// TIA Portal V17 export
// export: Created 2025-03-05T08:00:44.5361321Z, ExportSetting WithDefaults, DisplayName Totally Integrated Automation Portal, DisplayVersion V17 Update 8, DisplayName TIA Portal Openness, DisplayVersion V17 Update 8, DisplayName TIA Portal Version Control Interface, DisplayVersion V17, DisplayName SINAMICS Startdrive Advanced, DisplayVersion V17 SP2, DisplayName SINAMICS Startdrive G110M, G120, G120C, G120D, G120P, G115D, DisplayVersion V17 SP2, DisplayName SINAMICS Startdrive G130, G150, S120, S150, SINAMICS MV, S210, DisplayVersion V17 SP2, DisplayName STEP 7 Professional, DisplayVersion V17 Update 8, DisplayName SINUMERIK ONE STEP 7 Toolbox, DisplayVersion V17 Update 12, DisplayName SINUMERIK 840D sl STEP 7 Toolbox, DisplayVersion V17 Update 12, DisplayName STEP 7 Safety, DisplayVersion V17 Update 6, DisplayName WinCC Advanced, DisplayVersion V17 Update 8
FUNCTION "FC1314_UNIT_03_MASTER_MEASUREMENT" : Void   // FC1314, LAD
{ S7_Optimized_Access := 'FALSE' }
AUTHOR : ETXETAR
VERSION : 1.0
// stored: AutoNumber false, IsIECCheckEnabled false, SetENOAutomatically false, UDAEnableTagReadback false
   VAR_TEMP
      UNIT_01_STATION_0_LOCAL_E_RETURNS : Bool;   // UNIT 01 STATION 0 LOCAL E RETURNS
      UNIT_01_STATION_0_MACHINE_E_RETURNS : Bool;   // UNIT 01 STATION 0 MACHINE E RETURNS
   END_VAR
   VAR CONSTANT
      FC_NUMBER : DInt := 1314;
   END_VAR
   VAR_TEMP   // added for the SCL form of the ladder/FBD networks
      _w1 : Bool;
   END_VAR
BEGIN

REGION Network 1: GENERAL CONDITIONS
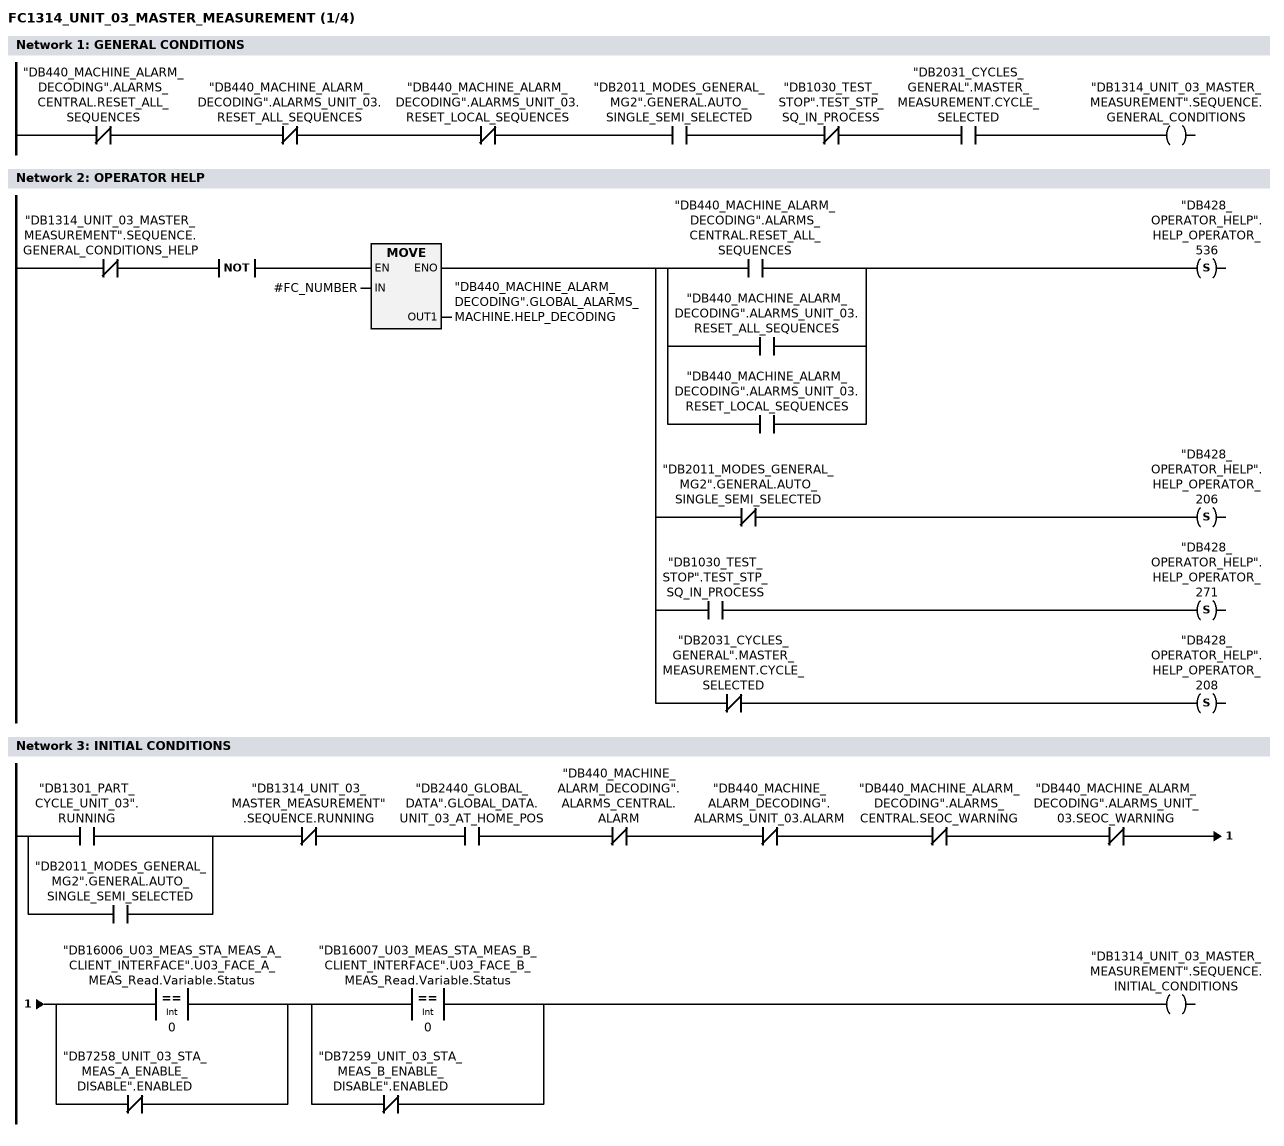
   RUNG wire#powerrail
      I_Contact( "DB440_MACHINE_ALARM_DECODING".ALARMS_CENTRAL.RESET_ALL_SEQUENCES )
      I_Contact( "DB440_MACHINE_ALARM_DECODING".ALARMS_UNIT_03.RESET_ALL_SEQUENCES )
      I_Contact( "DB440_MACHINE_ALARM_DECODING".ALARMS_UNIT_03.RESET_LOCAL_SEQUENCES )
      Contact( "DB2011_MODES_GENERAL_MG2".GENERAL.AUTO_SINGLE_SEMI_SELECTED )
      I_Contact( "DB1030_TEST_STOP".TEST_STP_SQ_IN_PROCESS )
      Contact( "DB2031_CYCLES_GENERAL".MASTER_MEASUREMENT.CYCLE_SELECTED )
      Coil( "DB1314_UNIT_03_MASTER_MEASUREMENT".SEQUENCE.GENERAL_CONDITIONS )
   END_RUNG
   // the same network as SCL:
   "DB1314_UNIT_03_MASTER_MEASUREMENT".SEQUENCE.GENERAL_CONDITIONS := NOT "DB440_MACHINE_ALARM_DECODING".ALARMS_CENTRAL.RESET_ALL_SEQUENCES AND NOT "DB440_MACHINE_ALARM_DECODING".ALARMS_UNIT_03.RESET_ALL_SEQUENCES AND NOT "DB440_MACHINE_ALARM_DECODING".ALARMS_UNIT_03.RESET_LOCAL_SEQUENCES AND "DB2011_MODES_GENERAL_MG2".GENERAL.AUTO_SINGLE_SEMI_SELECTED AND NOT "DB1030_TEST_STOP".TEST_STP_SQ_IN_PROCESS AND "DB2031_CYCLES_GENERAL".MASTER_MEASUREMENT.CYCLE_SELECTED;
END_REGION

REGION Network 2: OPERATOR HELP
   RUNG wire#powerrail
      I_Contact( "DB1314_UNIT_03_MASTER_MEASUREMENT".SEQUENCE.GENERAL_CONDITIONS_HELP )
      Not()
      { S7_GenerateENO := "TRUE" } Move(in := #FC_NUMBER, out1 => "DB440_MACHINE_ALARM_DECODING".GLOBAL_ALARMS_MACHINE.HELP_DECODING)
      wire#w1
      Contact( "DB440_MACHINE_ALARM_DECODING".ALARMS_CENTRAL.RESET_ALL_SEQUENCES )
      wire#w2
      S_Coil( "DB428_OPERATOR_HELP".HELP_OPERATOR_536 )
   END_RUNG
   RUNG wire#w1
      Contact( "DB440_MACHINE_ALARM_DECODING".ALARMS_UNIT_03.RESET_ALL_SEQUENCES )
   END_RUNG wire#w2
   RUNG wire#w1
      Contact( "DB440_MACHINE_ALARM_DECODING".ALARMS_UNIT_03.RESET_LOCAL_SEQUENCES )
   END_RUNG wire#w2
   RUNG wire#w1
      I_Contact( "DB2011_MODES_GENERAL_MG2".GENERAL.AUTO_SINGLE_SEMI_SELECTED )
      S_Coil( "DB428_OPERATOR_HELP".HELP_OPERATOR_206 )
   END_RUNG
   RUNG wire#w1
      Contact( "DB1030_TEST_STOP".TEST_STP_SQ_IN_PROCESS )
      S_Coil( "DB428_OPERATOR_HELP".HELP_OPERATOR_271 )
   END_RUNG
   RUNG wire#w1
      I_Contact( "DB2031_CYCLES_GENERAL".MASTER_MEASUREMENT.CYCLE_SELECTED )
      S_Coil( "DB428_OPERATOR_HELP".HELP_OPERATOR_208 )
   END_RUNG
   // the same network as SCL:
   // ENO of a box is taken as its EN; it also drops when the box reports an error
   #_w1 := NOT (NOT "DB1314_UNIT_03_MASTER_MEASUREMENT".SEQUENCE.GENERAL_CONDITIONS_HELP);
   IF #_w1 THEN "DB440_MACHINE_ALARM_DECODING".GLOBAL_ALARMS_MACHINE.HELP_DECODING := #FC_NUMBER; END_IF;
   IF #_w1 AND ("DB440_MACHINE_ALARM_DECODING".ALARMS_CENTRAL.RESET_ALL_SEQUENCES OR "DB440_MACHINE_ALARM_DECODING".ALARMS_UNIT_03.RESET_ALL_SEQUENCES OR "DB440_MACHINE_ALARM_DECODING".ALARMS_UNIT_03.RESET_LOCAL_SEQUENCES) THEN
       "DB428_OPERATOR_HELP".HELP_OPERATOR_536 := TRUE;
   END_IF;
   IF #_w1 AND NOT "DB2011_MODES_GENERAL_MG2".GENERAL.AUTO_SINGLE_SEMI_SELECTED THEN
       "DB428_OPERATOR_HELP".HELP_OPERATOR_206 := TRUE;
   END_IF;
   IF #_w1 AND "DB1030_TEST_STOP".TEST_STP_SQ_IN_PROCESS THEN
       "DB428_OPERATOR_HELP".HELP_OPERATOR_271 := TRUE;
   END_IF;
   IF #_w1 AND NOT "DB2031_CYCLES_GENERAL".MASTER_MEASUREMENT.CYCLE_SELECTED THEN
       "DB428_OPERATOR_HELP".HELP_OPERATOR_208 := TRUE;
   END_IF;
END_REGION

REGION Network 3: INITIAL CONDITIONS
   RUNG wire#powerrail
      Contact( "DB1301_PART_CYCLE_UNIT_03".RUNNING )
      wire#w1
      I_Contact( "DB1314_UNIT_03_MASTER_MEASUREMENT".SEQUENCE.RUNNING )
      Contact( "DB2440_GLOBAL_DATA".GLOBAL_DATA.UNIT_03_AT_HOME_POS )
      I_Contact( "DB440_MACHINE_ALARM_DECODING".ALARMS_CENTRAL.ALARM )
      I_Contact( "DB440_MACHINE_ALARM_DECODING".ALARMS_UNIT_03.ALARM )
      I_Contact( "DB440_MACHINE_ALARM_DECODING".ALARMS_CENTRAL.SEOC_WARNING )
      I_Contact( "DB440_MACHINE_ALARM_DECODING".ALARMS_UNIT_03.SEOC_WARNING )
      wire#w2
      { S7_Templates := "SrcType := Int" } EQ_Contact(in1 := "DB16006_U03_MEAS_STA_MEAS_A_CLIENT_INTERFACE".U03_FACE_A_MEAS_Read.Variable.Status, in2 := 0)
      wire#w3
      { S7_Templates := "SrcType := Int" } EQ_Contact(in1 := "DB16007_U03_MEAS_STA_MEAS_B_CLIENT_INTERFACE".U03_FACE_B_MEAS_Read.Variable.Status, in2 := 0)
      wire#w4
      Coil( "DB1314_UNIT_03_MASTER_MEASUREMENT".SEQUENCE.INITIAL_CONDITIONS )
   END_RUNG
   RUNG wire#powerrail
      Contact( "DB2011_MODES_GENERAL_MG2".GENERAL.AUTO_SINGLE_SEMI_SELECTED )
   END_RUNG wire#w1
   RUNG wire#w2
      I_Contact( "DB7258_UNIT_03_STA_MEAS_A_ENABLE_DISABLE".ENABLED )
   END_RUNG wire#w3
   RUNG wire#w3
      I_Contact( "DB7259_UNIT_03_STA_MEAS_B_ENABLE_DISABLE".ENABLED )
   END_RUNG wire#w4
   // the same network as SCL:
   "DB1314_UNIT_03_MASTER_MEASUREMENT".SEQUENCE.INITIAL_CONDITIONS := ("DB1301_PART_CYCLE_UNIT_03".RUNNING OR "DB2011_MODES_GENERAL_MG2".GENERAL.AUTO_SINGLE_SEMI_SELECTED) AND NOT "DB1314_UNIT_03_MASTER_MEASUREMENT".SEQUENCE.RUNNING AND "DB2440_GLOBAL_DATA".GLOBAL_DATA.UNIT_03_AT_HOME_POS AND NOT "DB440_MACHINE_ALARM_DECODING".ALARMS_CENTRAL.ALARM AND NOT "DB440_MACHINE_ALARM_DECODING".ALARMS_UNIT_03.ALARM AND NOT "DB440_MACHINE_ALARM_DECODING".ALARMS_CENTRAL.SEOC_WARNING AND NOT "DB440_MACHINE_ALARM_DECODING".ALARMS_UNIT_03.SEOC_WARNING AND (("DB16006_U03_MEAS_STA_MEAS_A_CLIENT_INTERFACE".U03_FACE_A_MEAS_Read.Variable.Status = 0) OR NOT "DB7258_UNIT_03_STA_MEAS_A_ENABLE_DISABLE".ENABLED) AND (("DB16007_U03_MEAS_STA_MEAS_B_CLIENT_INTERFACE".U03_FACE_B_MEAS_Read.Variable.Status = 0) OR NOT "DB7259_UNIT_03_STA_MEAS_B_ENABLE_DISABLE".ENABLED);
END_REGION

REGION Network 4: OPERATOR HELP
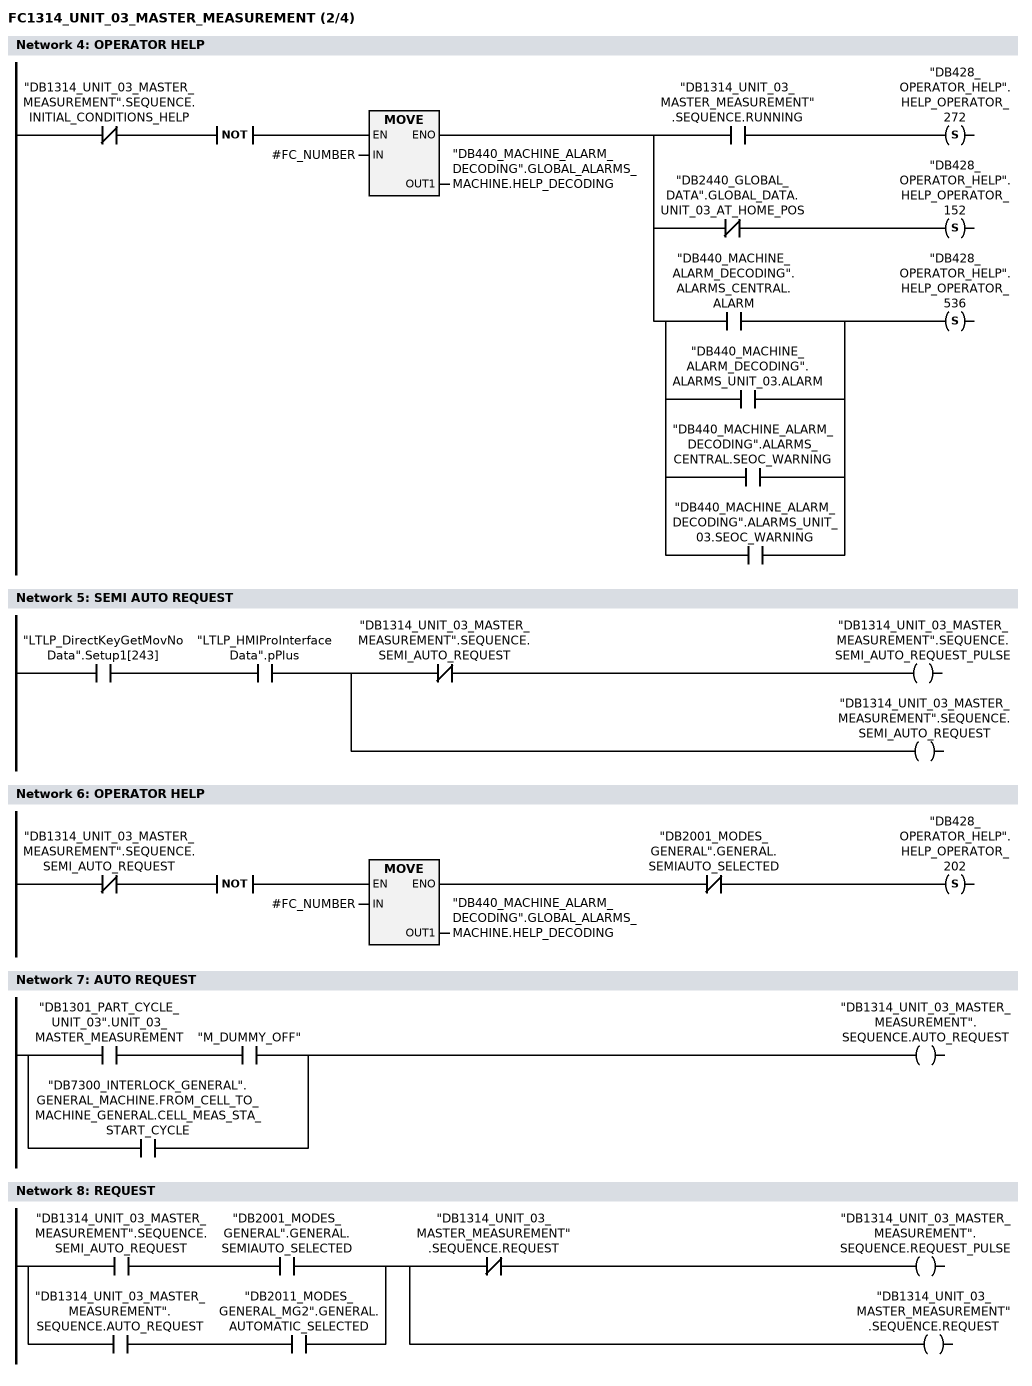
   RUNG wire#powerrail
      I_Contact( "DB1314_UNIT_03_MASTER_MEASUREMENT".SEQUENCE.INITIAL_CONDITIONS_HELP )
      Not()
      { S7_GenerateENO := "TRUE" } Move(in := #FC_NUMBER, out1 => "DB440_MACHINE_ALARM_DECODING".GLOBAL_ALARMS_MACHINE.HELP_DECODING)
      wire#w1
      Contact( "DB1314_UNIT_03_MASTER_MEASUREMENT".SEQUENCE.RUNNING )
      S_Coil( "DB428_OPERATOR_HELP".HELP_OPERATOR_272 )
   END_RUNG
   RUNG wire#w1
      I_Contact( "DB2440_GLOBAL_DATA".GLOBAL_DATA.UNIT_03_AT_HOME_POS )
      S_Coil( "DB428_OPERATOR_HELP".HELP_OPERATOR_152 )
   END_RUNG
   RUNG wire#w1
      Contact( "DB440_MACHINE_ALARM_DECODING".ALARMS_CENTRAL.ALARM )
      wire#w2
      S_Coil( "DB428_OPERATOR_HELP".HELP_OPERATOR_536 )
   END_RUNG
   RUNG wire#w1
      Contact( "DB440_MACHINE_ALARM_DECODING".ALARMS_UNIT_03.ALARM )
   END_RUNG wire#w2
   RUNG wire#w1
      Contact( "DB440_MACHINE_ALARM_DECODING".ALARMS_CENTRAL.SEOC_WARNING )
   END_RUNG wire#w2
   RUNG wire#w1
      Contact( "DB440_MACHINE_ALARM_DECODING".ALARMS_UNIT_03.SEOC_WARNING )
   END_RUNG wire#w2
   // the same network as SCL:
   // ENO of a box is taken as its EN; it also drops when the box reports an error
   #_w1 := NOT (NOT "DB1314_UNIT_03_MASTER_MEASUREMENT".SEQUENCE.INITIAL_CONDITIONS_HELP);
   IF #_w1 THEN "DB440_MACHINE_ALARM_DECODING".GLOBAL_ALARMS_MACHINE.HELP_DECODING := #FC_NUMBER; END_IF;
   IF #_w1 AND "DB1314_UNIT_03_MASTER_MEASUREMENT".SEQUENCE.RUNNING THEN
       "DB428_OPERATOR_HELP".HELP_OPERATOR_272 := TRUE;
   END_IF;
   IF #_w1 AND NOT "DB2440_GLOBAL_DATA".GLOBAL_DATA.UNIT_03_AT_HOME_POS THEN
       "DB428_OPERATOR_HELP".HELP_OPERATOR_152 := TRUE;
   END_IF;
   IF #_w1 AND ("DB440_MACHINE_ALARM_DECODING".ALARMS_CENTRAL.ALARM OR "DB440_MACHINE_ALARM_DECODING".ALARMS_UNIT_03.ALARM OR "DB440_MACHINE_ALARM_DECODING".ALARMS_CENTRAL.SEOC_WARNING OR "DB440_MACHINE_ALARM_DECODING".ALARMS_UNIT_03.SEOC_WARNING) THEN
       "DB428_OPERATOR_HELP".HELP_OPERATOR_536 := TRUE;
   END_IF;
END_REGION

REGION Network 5: SEMI AUTO REQUEST
   RUNG wire#powerrail
      Contact( "LTLP_DirectKeyGetMovNoData".Setup1[243] )
      Contact( "LTLP_HMIProInterfaceData".pPlus )
      wire#w1
      I_Contact( "DB1314_UNIT_03_MASTER_MEASUREMENT".SEQUENCE.SEMI_AUTO_REQUEST )
      Coil( "DB1314_UNIT_03_MASTER_MEASUREMENT".SEQUENCE.SEMI_AUTO_REQUEST_PULSE )
   END_RUNG
   RUNG wire#w1
      Coil( "DB1314_UNIT_03_MASTER_MEASUREMENT".SEQUENCE.SEMI_AUTO_REQUEST )
   END_RUNG
   // the same network as SCL:
   #_w1 := "LTLP_DirectKeyGetMovNoData".Setup1[243] AND "LTLP_HMIProInterfaceData".pPlus;
   "DB1314_UNIT_03_MASTER_MEASUREMENT".SEQUENCE.SEMI_AUTO_REQUEST_PULSE := #_w1 AND NOT "DB1314_UNIT_03_MASTER_MEASUREMENT".SEQUENCE.SEMI_AUTO_REQUEST;
   "DB1314_UNIT_03_MASTER_MEASUREMENT".SEQUENCE.SEMI_AUTO_REQUEST := #_w1;
END_REGION

REGION Network 6: OPERATOR HELP
   RUNG wire#powerrail
      I_Contact( "DB1314_UNIT_03_MASTER_MEASUREMENT".SEQUENCE.SEMI_AUTO_REQUEST )
      Not()
      { S7_GenerateENO := "TRUE" } Move(in := #FC_NUMBER, out1 => "DB440_MACHINE_ALARM_DECODING".GLOBAL_ALARMS_MACHINE.HELP_DECODING)
      I_Contact( "DB2001_MODES_GENERAL".GENERAL.SEMIAUTO_SELECTED )
      S_Coil( "DB428_OPERATOR_HELP".HELP_OPERATOR_202 )
   END_RUNG
   // the same network as SCL:
   // ENO of a box is taken as its EN; it also drops when the box reports an error
   #_w1 := NOT (NOT "DB1314_UNIT_03_MASTER_MEASUREMENT".SEQUENCE.SEMI_AUTO_REQUEST);
   IF #_w1 THEN "DB440_MACHINE_ALARM_DECODING".GLOBAL_ALARMS_MACHINE.HELP_DECODING := #FC_NUMBER; END_IF;
   IF #_w1 AND NOT "DB2001_MODES_GENERAL".GENERAL.SEMIAUTO_SELECTED THEN
       "DB428_OPERATOR_HELP".HELP_OPERATOR_202 := TRUE;
   END_IF;
END_REGION

REGION Network 7: AUTO REQUEST
   RUNG wire#powerrail
      Contact( "DB1301_PART_CYCLE_UNIT_03".UNIT_03_MASTER_MEASUREMENT )
      Contact( "M_DUMMY_OFF" )
      wire#w1
      Coil( "DB1314_UNIT_03_MASTER_MEASUREMENT".SEQUENCE.AUTO_REQUEST )
   END_RUNG
   RUNG wire#powerrail
      Contact( "DB7300_INTERLOCK_GENERAL".GENERAL_MACHINE.FROM_CELL_TO_MACHINE_GENERAL.CELL_MEAS_STA_START_CYCLE )
   END_RUNG wire#w1
   // the same network as SCL:
   "DB1314_UNIT_03_MASTER_MEASUREMENT".SEQUENCE.AUTO_REQUEST := ("DB1301_PART_CYCLE_UNIT_03".UNIT_03_MASTER_MEASUREMENT AND "M_DUMMY_OFF") OR "DB7300_INTERLOCK_GENERAL".GENERAL_MACHINE.FROM_CELL_TO_MACHINE_GENERAL.CELL_MEAS_STA_START_CYCLE;
END_REGION

REGION Network 8: REQUEST
   RUNG wire#powerrail
      Contact( "DB1314_UNIT_03_MASTER_MEASUREMENT".SEQUENCE.SEMI_AUTO_REQUEST )
      Contact( "DB2001_MODES_GENERAL".GENERAL.SEMIAUTO_SELECTED )
      wire#w1
      I_Contact( "DB1314_UNIT_03_MASTER_MEASUREMENT".SEQUENCE.REQUEST )
      Coil( "DB1314_UNIT_03_MASTER_MEASUREMENT".SEQUENCE.REQUEST_PULSE )
   END_RUNG
   RUNG wire#powerrail
      Contact( "DB1314_UNIT_03_MASTER_MEASUREMENT".SEQUENCE.AUTO_REQUEST )
      Contact( "DB2011_MODES_GENERAL_MG2".GENERAL.AUTOMATIC_SELECTED )
   END_RUNG wire#w1
   RUNG wire#w1
      Coil( "DB1314_UNIT_03_MASTER_MEASUREMENT".SEQUENCE.REQUEST )
   END_RUNG
   // the same network as SCL:
   #_w1 := ("DB1314_UNIT_03_MASTER_MEASUREMENT".SEQUENCE.SEMI_AUTO_REQUEST AND "DB2001_MODES_GENERAL".GENERAL.SEMIAUTO_SELECTED) OR ("DB1314_UNIT_03_MASTER_MEASUREMENT".SEQUENCE.AUTO_REQUEST AND "DB2011_MODES_GENERAL_MG2".GENERAL.AUTOMATIC_SELECTED);
   "DB1314_UNIT_03_MASTER_MEASUREMENT".SEQUENCE.REQUEST_PULSE := #_w1 AND NOT "DB1314_UNIT_03_MASTER_MEASUREMENT".SEQUENCE.REQUEST;
   "DB1314_UNIT_03_MASTER_MEASUREMENT".SEQUENCE.REQUEST := #_w1;
END_REGION

REGION Network 9: COMMAND
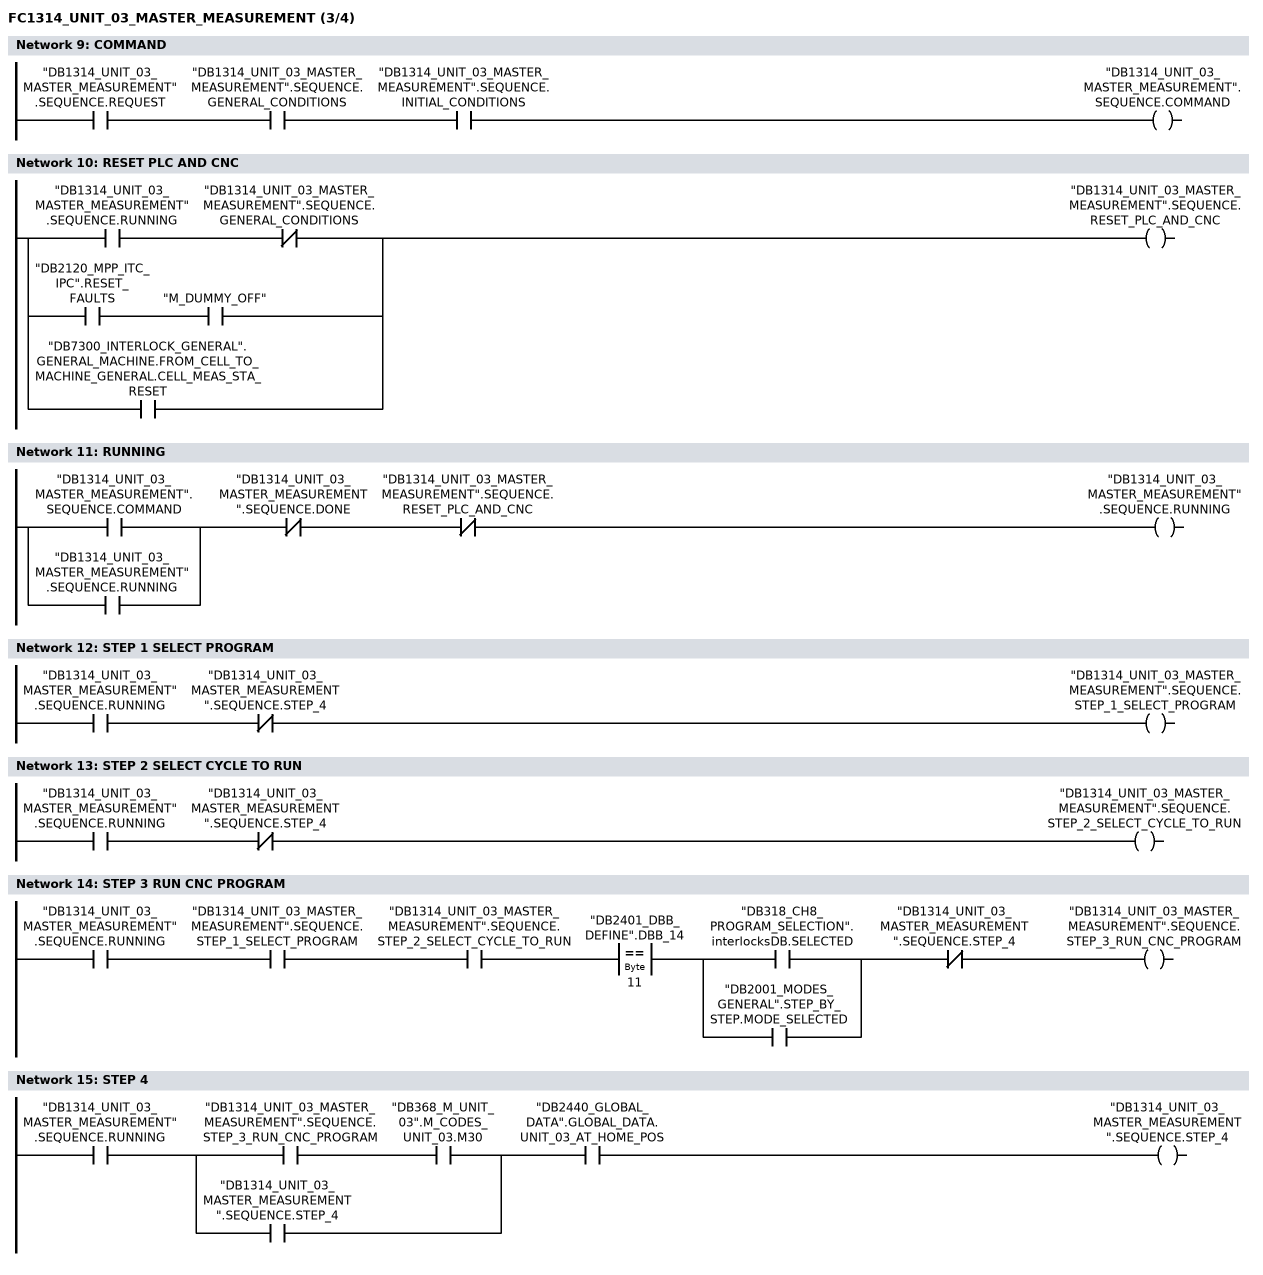
   RUNG wire#powerrail
      Contact( "DB1314_UNIT_03_MASTER_MEASUREMENT".SEQUENCE.REQUEST )
      Contact( "DB1314_UNIT_03_MASTER_MEASUREMENT".SEQUENCE.GENERAL_CONDITIONS )
      Contact( "DB1314_UNIT_03_MASTER_MEASUREMENT".SEQUENCE.INITIAL_CONDITIONS )
      Coil( "DB1314_UNIT_03_MASTER_MEASUREMENT".SEQUENCE.COMMAND )
   END_RUNG
   // the same network as SCL:
   "DB1314_UNIT_03_MASTER_MEASUREMENT".SEQUENCE.COMMAND := "DB1314_UNIT_03_MASTER_MEASUREMENT".SEQUENCE.REQUEST AND "DB1314_UNIT_03_MASTER_MEASUREMENT".SEQUENCE.GENERAL_CONDITIONS AND "DB1314_UNIT_03_MASTER_MEASUREMENT".SEQUENCE.INITIAL_CONDITIONS;
END_REGION

REGION Network 10: RESET PLC AND CNC
   RUNG wire#powerrail
      Contact( "DB1314_UNIT_03_MASTER_MEASUREMENT".SEQUENCE.RUNNING )
      I_Contact( "DB1314_UNIT_03_MASTER_MEASUREMENT".SEQUENCE.GENERAL_CONDITIONS )
      wire#w1
      Coil( "DB1314_UNIT_03_MASTER_MEASUREMENT".SEQUENCE.RESET_PLC_AND_CNC )
   END_RUNG
   RUNG wire#powerrail
      Contact( "DB2120_MPP_ITC_IPC".RESET_FAULTS )
      Contact( "M_DUMMY_OFF" )
   END_RUNG wire#w1
   RUNG wire#powerrail
      Contact( "DB7300_INTERLOCK_GENERAL".GENERAL_MACHINE.FROM_CELL_TO_MACHINE_GENERAL.CELL_MEAS_STA_RESET )
   END_RUNG wire#w1
   // the same network as SCL:
   "DB1314_UNIT_03_MASTER_MEASUREMENT".SEQUENCE.RESET_PLC_AND_CNC := ("DB1314_UNIT_03_MASTER_MEASUREMENT".SEQUENCE.RUNNING AND NOT "DB1314_UNIT_03_MASTER_MEASUREMENT".SEQUENCE.GENERAL_CONDITIONS) OR ("DB2120_MPP_ITC_IPC".RESET_FAULTS AND "M_DUMMY_OFF") OR "DB7300_INTERLOCK_GENERAL".GENERAL_MACHINE.FROM_CELL_TO_MACHINE_GENERAL.CELL_MEAS_STA_RESET;
END_REGION

REGION Network 11: RUNNING
   RUNG wire#powerrail
      Contact( "DB1314_UNIT_03_MASTER_MEASUREMENT".SEQUENCE.COMMAND )
      wire#w1
      I_Contact( "DB1314_UNIT_03_MASTER_MEASUREMENT".SEQUENCE.DONE )
      I_Contact( "DB1314_UNIT_03_MASTER_MEASUREMENT".SEQUENCE.RESET_PLC_AND_CNC )
      Coil( "DB1314_UNIT_03_MASTER_MEASUREMENT".SEQUENCE.RUNNING )
   END_RUNG
   RUNG wire#powerrail
      Contact( "DB1314_UNIT_03_MASTER_MEASUREMENT".SEQUENCE.RUNNING )
   END_RUNG wire#w1
   // the same network as SCL:
   "DB1314_UNIT_03_MASTER_MEASUREMENT".SEQUENCE.RUNNING := ("DB1314_UNIT_03_MASTER_MEASUREMENT".SEQUENCE.COMMAND OR "DB1314_UNIT_03_MASTER_MEASUREMENT".SEQUENCE.RUNNING) AND NOT "DB1314_UNIT_03_MASTER_MEASUREMENT".SEQUENCE.DONE AND NOT "DB1314_UNIT_03_MASTER_MEASUREMENT".SEQUENCE.RESET_PLC_AND_CNC;
END_REGION

REGION Network 12: STEP 1 SELECT PROGRAM
   RUNG wire#powerrail
      Contact( "DB1314_UNIT_03_MASTER_MEASUREMENT".SEQUENCE.RUNNING )
      I_Contact( "DB1314_UNIT_03_MASTER_MEASUREMENT".SEQUENCE.STEP_4 )
      Coil( "DB1314_UNIT_03_MASTER_MEASUREMENT".SEQUENCE.STEP_1_SELECT_PROGRAM )
   END_RUNG
   // the same network as SCL:
   "DB1314_UNIT_03_MASTER_MEASUREMENT".SEQUENCE.STEP_1_SELECT_PROGRAM := "DB1314_UNIT_03_MASTER_MEASUREMENT".SEQUENCE.RUNNING AND NOT "DB1314_UNIT_03_MASTER_MEASUREMENT".SEQUENCE.STEP_4;
END_REGION

REGION Network 13: STEP 2 SELECT CYCLE TO RUN
   RUNG wire#powerrail
      Contact( "DB1314_UNIT_03_MASTER_MEASUREMENT".SEQUENCE.RUNNING )
      I_Contact( "DB1314_UNIT_03_MASTER_MEASUREMENT".SEQUENCE.STEP_4 )
      Coil( "DB1314_UNIT_03_MASTER_MEASUREMENT".SEQUENCE.STEP_2_SELECT_CYCLE_TO_RUN )
   END_RUNG
   // the same network as SCL:
   "DB1314_UNIT_03_MASTER_MEASUREMENT".SEQUENCE.STEP_2_SELECT_CYCLE_TO_RUN := "DB1314_UNIT_03_MASTER_MEASUREMENT".SEQUENCE.RUNNING AND NOT "DB1314_UNIT_03_MASTER_MEASUREMENT".SEQUENCE.STEP_4;
END_REGION

REGION Network 14: STEP 3 RUN CNC PROGRAM
   RUNG wire#powerrail
      Contact( "DB1314_UNIT_03_MASTER_MEASUREMENT".SEQUENCE.RUNNING )
      Contact( "DB1314_UNIT_03_MASTER_MEASUREMENT".SEQUENCE.STEP_1_SELECT_PROGRAM )
      Contact( "DB1314_UNIT_03_MASTER_MEASUREMENT".SEQUENCE.STEP_2_SELECT_CYCLE_TO_RUN )
      { S7_Templates := "SrcType := Byte" } EQ_Contact(in1 := "DB2401_DBB_DEFINE".DBB_14, in2 := 11)
      wire#w1
      Contact( "DB318_CH8_PROGRAM_SELECTION".interlocksDB.SELECTED )
      wire#w2
      I_Contact( "DB1314_UNIT_03_MASTER_MEASUREMENT".SEQUENCE.STEP_4 )
      Coil( "DB1314_UNIT_03_MASTER_MEASUREMENT".SEQUENCE.STEP_3_RUN_CNC_PROGRAM )
   END_RUNG
   RUNG wire#w1
      Contact( "DB2001_MODES_GENERAL".STEP_BY_STEP.MODE_SELECTED )
   END_RUNG wire#w2
   // the same network as SCL:
   "DB1314_UNIT_03_MASTER_MEASUREMENT".SEQUENCE.STEP_3_RUN_CNC_PROGRAM := "DB1314_UNIT_03_MASTER_MEASUREMENT".SEQUENCE.RUNNING AND "DB1314_UNIT_03_MASTER_MEASUREMENT".SEQUENCE.STEP_1_SELECT_PROGRAM AND "DB1314_UNIT_03_MASTER_MEASUREMENT".SEQUENCE.STEP_2_SELECT_CYCLE_TO_RUN AND ("DB2401_DBB_DEFINE".DBB_14 = 11) AND ("DB318_CH8_PROGRAM_SELECTION".interlocksDB.SELECTED OR "DB2001_MODES_GENERAL".STEP_BY_STEP.MODE_SELECTED) AND NOT "DB1314_UNIT_03_MASTER_MEASUREMENT".SEQUENCE.STEP_4;
END_REGION

REGION Network 15: STEP 4
   RUNG wire#powerrail
      Contact( "DB1314_UNIT_03_MASTER_MEASUREMENT".SEQUENCE.RUNNING )
      wire#w1
      Contact( "DB1314_UNIT_03_MASTER_MEASUREMENT".SEQUENCE.STEP_3_RUN_CNC_PROGRAM )
      Contact( "DB368_M_UNIT_03".M_CODES_UNIT_03.M30 )
      wire#w2
      Contact( "DB2440_GLOBAL_DATA".GLOBAL_DATA.UNIT_03_AT_HOME_POS )
      Coil( "DB1314_UNIT_03_MASTER_MEASUREMENT".SEQUENCE.STEP_4 )
   END_RUNG
   RUNG wire#w1
      Contact( "DB1314_UNIT_03_MASTER_MEASUREMENT".SEQUENCE.STEP_4 )
   END_RUNG wire#w2
   // the same network as SCL:
   "DB1314_UNIT_03_MASTER_MEASUREMENT".SEQUENCE.STEP_4 := "DB1314_UNIT_03_MASTER_MEASUREMENT".SEQUENCE.RUNNING AND (("DB1314_UNIT_03_MASTER_MEASUREMENT".SEQUENCE.STEP_3_RUN_CNC_PROGRAM AND "DB368_M_UNIT_03".M_CODES_UNIT_03.M30) OR "DB1314_UNIT_03_MASTER_MEASUREMENT".SEQUENCE.STEP_4) AND "DB2440_GLOBAL_DATA".GLOBAL_DATA.UNIT_03_AT_HOME_POS;
END_REGION

REGION Network 16: DONE
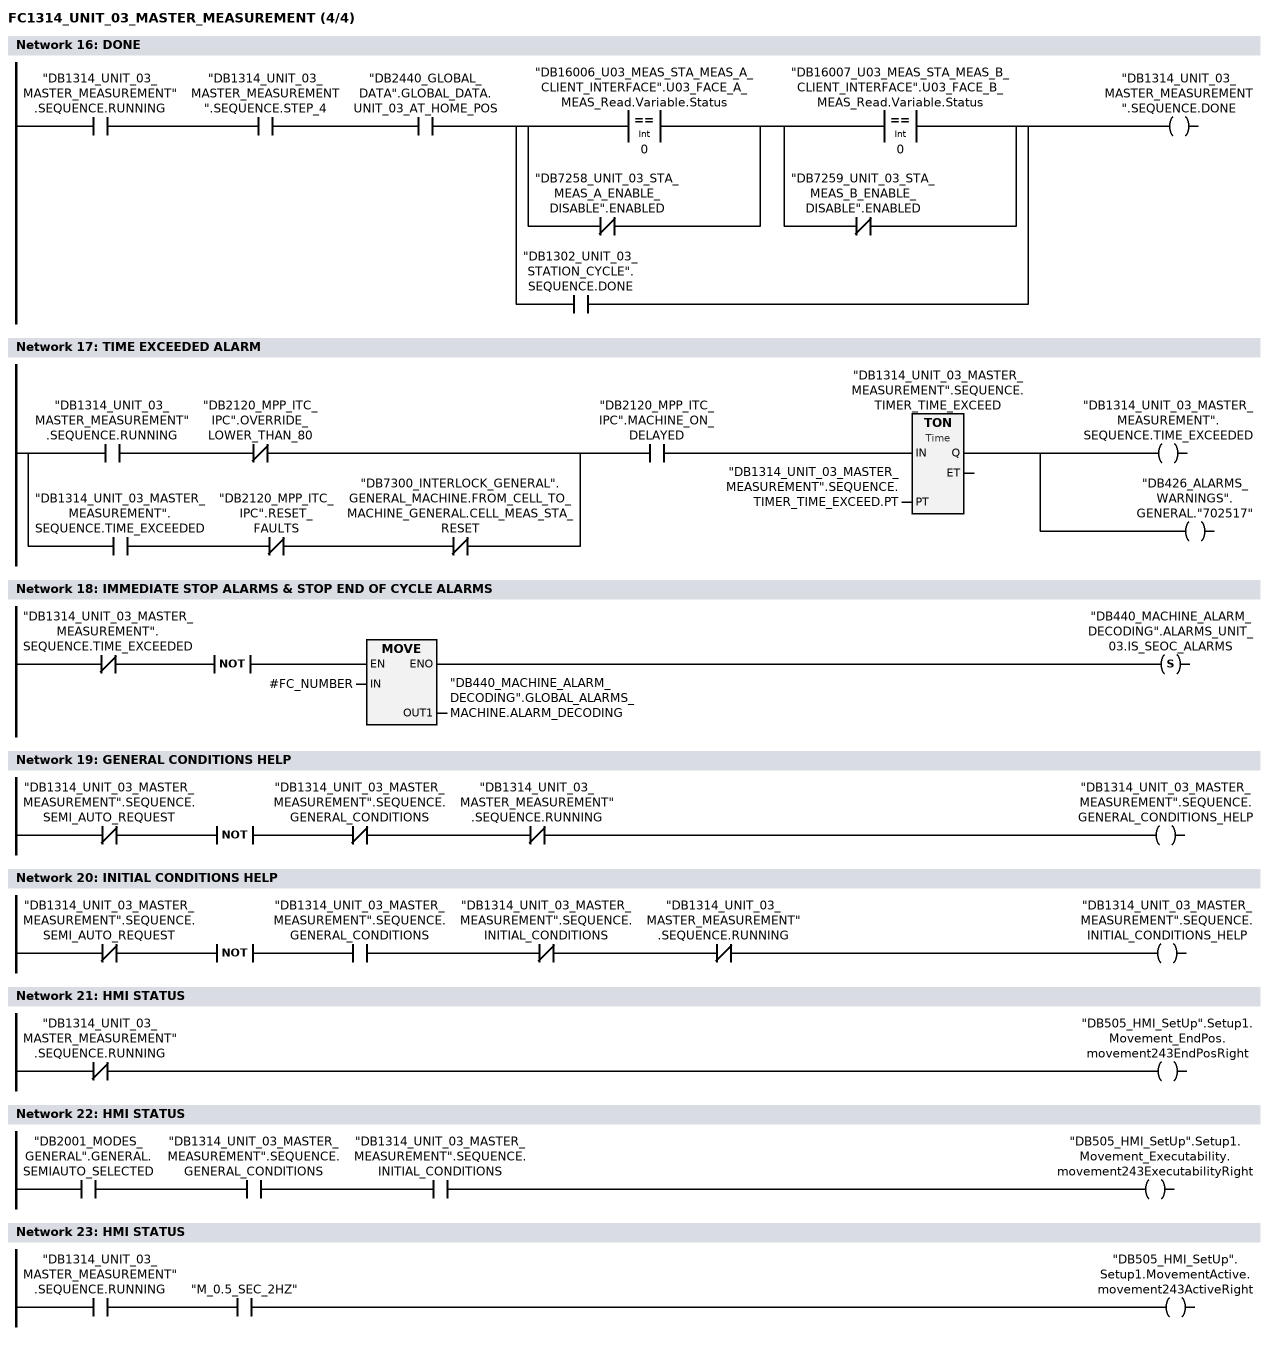
   RUNG wire#powerrail
      Contact( "DB1314_UNIT_03_MASTER_MEASUREMENT".SEQUENCE.RUNNING )
      Contact( "DB1314_UNIT_03_MASTER_MEASUREMENT".SEQUENCE.STEP_4 )
      Contact( "DB2440_GLOBAL_DATA".GLOBAL_DATA.UNIT_03_AT_HOME_POS )
      wire#w1
      { S7_Templates := "SrcType := Int" } EQ_Contact(in1 := "DB16006_U03_MEAS_STA_MEAS_A_CLIENT_INTERFACE".U03_FACE_A_MEAS_Read.Variable.Status, in2 := 0)
      wire#w2
      { S7_Templates := "SrcType := Int" } EQ_Contact(in1 := "DB16007_U03_MEAS_STA_MEAS_B_CLIENT_INTERFACE".U03_FACE_B_MEAS_Read.Variable.Status, in2 := 0)
      wire#w3
      Coil( "DB1314_UNIT_03_MASTER_MEASUREMENT".SEQUENCE.DONE )
   END_RUNG
   RUNG wire#w1
      I_Contact( "DB7258_UNIT_03_STA_MEAS_A_ENABLE_DISABLE".ENABLED )
   END_RUNG wire#w2
   RUNG wire#w2
      I_Contact( "DB7259_UNIT_03_STA_MEAS_B_ENABLE_DISABLE".ENABLED )
   END_RUNG wire#w3
   RUNG wire#w1
      Contact( "DB1302_UNIT_03_STATION_CYCLE".SEQUENCE.DONE )
   END_RUNG wire#w3
   // the same network as SCL:
   "DB1314_UNIT_03_MASTER_MEASUREMENT".SEQUENCE.DONE := "DB1314_UNIT_03_MASTER_MEASUREMENT".SEQUENCE.RUNNING AND "DB1314_UNIT_03_MASTER_MEASUREMENT".SEQUENCE.STEP_4 AND "DB2440_GLOBAL_DATA".GLOBAL_DATA.UNIT_03_AT_HOME_POS AND (((("DB16006_U03_MEAS_STA_MEAS_A_CLIENT_INTERFACE".U03_FACE_A_MEAS_Read.Variable.Status = 0) OR NOT "DB7258_UNIT_03_STA_MEAS_A_ENABLE_DISABLE".ENABLED) AND (("DB16007_U03_MEAS_STA_MEAS_B_CLIENT_INTERFACE".U03_FACE_B_MEAS_Read.Variable.Status = 0) OR NOT "DB7259_UNIT_03_STA_MEAS_B_ENABLE_DISABLE".ENABLED)) OR "DB1302_UNIT_03_STATION_CYCLE".SEQUENCE.DONE);
END_REGION

REGION Network 17: TIME EXCEEDED ALARM
   RUNG wire#powerrail
      Contact( "DB1314_UNIT_03_MASTER_MEASUREMENT".SEQUENCE.RUNNING )
      I_Contact( "DB2120_MPP_ITC_IPC".OVERRIDE_LOWER_THAN_80 )
      wire#w1
      Contact( "DB2120_MPP_ITC_IPC".MACHINE_ON_DELAYED )
      { S7_Templates := "time_type := Time" } "DB1314_UNIT_03_MASTER_MEASUREMENT".SEQUENCE.TIMER_TIME_EXCEED.TON(pt := "DB1314_UNIT_03_MASTER_MEASUREMENT".SEQUENCE.TIMER_TIME_EXCEED.PT, et =>)
      wire#w2
      Coil( "DB1314_UNIT_03_MASTER_MEASUREMENT".SEQUENCE.TIME_EXCEEDED )
   END_RUNG
   RUNG wire#powerrail
      Contact( "DB1314_UNIT_03_MASTER_MEASUREMENT".SEQUENCE.TIME_EXCEEDED )
      I_Contact( "DB2120_MPP_ITC_IPC".RESET_FAULTS )
      I_Contact( "DB7300_INTERLOCK_GENERAL".GENERAL_MACHINE.FROM_CELL_TO_MACHINE_GENERAL.CELL_MEAS_STA_RESET )
   END_RUNG wire#w1
   RUNG wire#w2
      Coil( "DB426_ALARMS_WARNINGS".GENERAL."702517" )
   END_RUNG
   // the same network as SCL:
   "DB1314_UNIT_03_MASTER_MEASUREMENT".SEQUENCE.TIMER_TIME_EXCEED.TON(IN := (("DB1314_UNIT_03_MASTER_MEASUREMENT".SEQUENCE.RUNNING AND NOT "DB2120_MPP_ITC_IPC".OVERRIDE_LOWER_THAN_80) OR ("DB1314_UNIT_03_MASTER_MEASUREMENT".SEQUENCE.TIME_EXCEEDED AND NOT "DB2120_MPP_ITC_IPC".RESET_FAULTS AND NOT "DB7300_INTERLOCK_GENERAL".GENERAL_MACHINE.FROM_CELL_TO_MACHINE_GENERAL.CELL_MEAS_STA_RESET)) AND "DB2120_MPP_ITC_IPC".MACHINE_ON_DELAYED,
                           PT := "DB1314_UNIT_03_MASTER_MEASUREMENT".SEQUENCE.TIMER_TIME_EXCEED.PT);
   "DB1314_UNIT_03_MASTER_MEASUREMENT".SEQUENCE.TIME_EXCEEDED := "DB1314_UNIT_03_MASTER_MEASUREMENT".SEQUENCE.TIMER_TIME_EXCEED.Q;
   "DB426_ALARMS_WARNINGS".GENERAL."702517" := "DB1314_UNIT_03_MASTER_MEASUREMENT".SEQUENCE.TIMER_TIME_EXCEED.Q;
END_REGION

REGION Network 18: IMMEDIATE STOP ALARMS & STOP END OF CYCLE ALARMS
   RUNG wire#powerrail
      I_Contact( "DB1314_UNIT_03_MASTER_MEASUREMENT".SEQUENCE.TIME_EXCEEDED )
      Not()
      { S7_GenerateENO := "TRUE" } Move(in := #FC_NUMBER, out1 => "DB440_MACHINE_ALARM_DECODING".GLOBAL_ALARMS_MACHINE.ALARM_DECODING)
      S_Coil( "DB440_MACHINE_ALARM_DECODING".ALARMS_UNIT_03.IS_SEOC_ALARMS )
   END_RUNG
   // the same network as SCL:
   // ENO of a box is taken as its EN; it also drops when the box reports an error
   IF NOT (NOT "DB1314_UNIT_03_MASTER_MEASUREMENT".SEQUENCE.TIME_EXCEEDED) THEN
       "DB440_MACHINE_ALARM_DECODING".GLOBAL_ALARMS_MACHINE.ALARM_DECODING := #FC_NUMBER;
       "DB440_MACHINE_ALARM_DECODING".ALARMS_UNIT_03.IS_SEOC_ALARMS := TRUE;
   END_IF;
END_REGION

REGION Network 19: GENERAL CONDITIONS HELP
   RUNG wire#powerrail
      I_Contact( "DB1314_UNIT_03_MASTER_MEASUREMENT".SEQUENCE.SEMI_AUTO_REQUEST )
      Not()
      I_Contact( "DB1314_UNIT_03_MASTER_MEASUREMENT".SEQUENCE.GENERAL_CONDITIONS )
      I_Contact( "DB1314_UNIT_03_MASTER_MEASUREMENT".SEQUENCE.RUNNING )
      Coil( "DB1314_UNIT_03_MASTER_MEASUREMENT".SEQUENCE.GENERAL_CONDITIONS_HELP )
   END_RUNG
   // the same network as SCL:
   "DB1314_UNIT_03_MASTER_MEASUREMENT".SEQUENCE.GENERAL_CONDITIONS_HELP := NOT (NOT "DB1314_UNIT_03_MASTER_MEASUREMENT".SEQUENCE.SEMI_AUTO_REQUEST) AND NOT "DB1314_UNIT_03_MASTER_MEASUREMENT".SEQUENCE.GENERAL_CONDITIONS AND NOT "DB1314_UNIT_03_MASTER_MEASUREMENT".SEQUENCE.RUNNING;
END_REGION

REGION Network 20: INITIAL CONDITIONS HELP
   RUNG wire#powerrail
      I_Contact( "DB1314_UNIT_03_MASTER_MEASUREMENT".SEQUENCE.SEMI_AUTO_REQUEST )
      Not()
      Contact( "DB1314_UNIT_03_MASTER_MEASUREMENT".SEQUENCE.GENERAL_CONDITIONS )
      I_Contact( "DB1314_UNIT_03_MASTER_MEASUREMENT".SEQUENCE.INITIAL_CONDITIONS )
      I_Contact( "DB1314_UNIT_03_MASTER_MEASUREMENT".SEQUENCE.RUNNING )
      Coil( "DB1314_UNIT_03_MASTER_MEASUREMENT".SEQUENCE.INITIAL_CONDITIONS_HELP )
   END_RUNG
   // the same network as SCL:
   "DB1314_UNIT_03_MASTER_MEASUREMENT".SEQUENCE.INITIAL_CONDITIONS_HELP := NOT (NOT "DB1314_UNIT_03_MASTER_MEASUREMENT".SEQUENCE.SEMI_AUTO_REQUEST) AND "DB1314_UNIT_03_MASTER_MEASUREMENT".SEQUENCE.GENERAL_CONDITIONS AND NOT "DB1314_UNIT_03_MASTER_MEASUREMENT".SEQUENCE.INITIAL_CONDITIONS AND NOT "DB1314_UNIT_03_MASTER_MEASUREMENT".SEQUENCE.RUNNING;
END_REGION

REGION Network 21: HMI STATUS
   RUNG wire#powerrail
      I_Contact( "DB1314_UNIT_03_MASTER_MEASUREMENT".SEQUENCE.RUNNING )
      Coil( "DB505_HMI_SetUp".Setup1.Movement_EndPos.movement243EndPosRight )
   END_RUNG
   // the same network as SCL:
   "DB505_HMI_SetUp".Setup1.Movement_EndPos.movement243EndPosRight := NOT "DB1314_UNIT_03_MASTER_MEASUREMENT".SEQUENCE.RUNNING;
END_REGION

REGION Network 22: HMI STATUS
   RUNG wire#powerrail
      Contact( "DB2001_MODES_GENERAL".GENERAL.SEMIAUTO_SELECTED )
      Contact( "DB1314_UNIT_03_MASTER_MEASUREMENT".SEQUENCE.GENERAL_CONDITIONS )
      Contact( "DB1314_UNIT_03_MASTER_MEASUREMENT".SEQUENCE.INITIAL_CONDITIONS )
      Coil( "DB505_HMI_SetUp".Setup1.Movement_Executability.movement243ExecutabilityRight )
   END_RUNG
   // the same network as SCL:
   "DB505_HMI_SetUp".Setup1.Movement_Executability.movement243ExecutabilityRight := "DB2001_MODES_GENERAL".GENERAL.SEMIAUTO_SELECTED AND "DB1314_UNIT_03_MASTER_MEASUREMENT".SEQUENCE.GENERAL_CONDITIONS AND "DB1314_UNIT_03_MASTER_MEASUREMENT".SEQUENCE.INITIAL_CONDITIONS;
END_REGION

REGION Network 23: HMI STATUS
   RUNG wire#powerrail
      Contact( "DB1314_UNIT_03_MASTER_MEASUREMENT".SEQUENCE.RUNNING )
      Contact( "M_0.5_SEC_2HZ" )
      Coil( "DB505_HMI_SetUp".Setup1.MovementActive.movement243ActiveRight )
   END_RUNG
   // the same network as SCL:
   "DB505_HMI_SetUp".Setup1.MovementActive.movement243ActiveRight := "DB1314_UNIT_03_MASTER_MEASUREMENT".SEQUENCE.RUNNING AND "M_0.5_SEC_2HZ";
END_REGION
END_FUNCTION
